// TwinCAT 3 PLC project task1
// ProgramVersion: 3.1.4022.4
// libraries:
//   Tc2_Standard, * (Beckhoff Automation GmbH)
//   Tc2_System, * (Beckhoff Automation GmbH)
//   Tc3_Module, * (Beckhoff Automation GmbH)
// project tree:
//   / PlcTask.TcTTO
//   POUs/ FB1.TcPOU, FB2.TcPOU, FB3.TcPOU, FB4.TcPOU, iFb.TcIO, MAIN.TcPOU
// real-time tasks:
//   TASK PlcTask: cycle T#10ms, priority 20, ADS port 350

CONFIGURATION task1
    RESOURCE PLC ON TwinCAT3
        TASK PlcTask(INTERVAL := T#10ms, PRIORITY := 20);
    END_RESOURCE
END_CONFIGURATION

// ---- POUs/iFb.TcIO
//Contiene due proprietà che sono i valori di input
//ed un metodo generico che calcola il valore
INTERFACE iFb

PROPERTY PUBLIC fInput1 : REAL
GET
END_GET
SET
END_SET
END_PROPERTY

PROPERTY PUBLIC fInput2 : REAL
GET
END_GET
SET
END_SET
END_PROPERTY

METHOD returnValue : REAL
VAR_INPUT
END_VAR
END_METHOD

END_INTERFACE

// ---- POUs/FB1.TcPOU
//La FB1 Implementa l'interfaccia iFB

FUNCTION_BLOCK PUBLIC FB1 IMPLEMENTS iFb
VAR_INPUT
END_VAR
VAR_OUTPUT
END_VAR
VAR
	fInternalInput1 : REAL;
	fInternalInput2 : REAL;
END_VAR

;

{warning 'add property implementation'}
PROPERTY fInput1 : REAL
GET
fInput1 := this^.fInternalInput1;
END_GET
SET
this^.fInternalInput1 := fInput1;
END_SET
END_PROPERTY

{warning 'add property implementation'}
PROPERTY fInput2 : REAL
GET
fInput2 := this^.fInternalInput2;
END_GET
SET
this^.fInternalInput2 := fInput2;
END_SET
END_PROPERTY

{warning 'add method implementation'}
METHOD returnValue : REAL
//Implementazione Interfaccia con somma
returnValue := this^.fInput1 + this^.fInput2;
END_METHOD

END_FUNCTION_BLOCK

// ---- POUs/FB2.TcPOU
//Anche FB2 Implementa l'interfaccia iFB
//Posso considerarla come un'altra implementazione della stessa

FUNCTION_BLOCK PUBLIC FB2 IMPLEMENTS iFb
VAR_INPUT
END_VAR
VAR_OUTPUT
END_VAR
VAR
	fInternalInput1 : REAL;
	fInternalInput2 : REAL;
END_VAR

{warning 'add property implementation'}
PROPERTY fInput1 : REAL
GET
fInput1 := this^.fInternalInput1;
END_GET
SET
this^.fInternalInput1 := fInput1;
END_SET
END_PROPERTY

{warning 'add property implementation'}
PROPERTY fInput2 : REAL
GET
fInput2 := this^.fInternalInput2;
END_GET
SET
this^.fInternalInput2 := fInput2;
END_SET
END_PROPERTY

{warning 'add method implementation'}
METHOD returnValue : REAL
//Implementazione Interfaccia con moltiplicazione
returnValue := this^.fInput1 * this^.fInput2;
END_METHOD

END_FUNCTION_BLOCK

// ---- POUs/FB3.TcPOU
//La FB3 estende la FB1 quindi anche lei implementa l'interfaccia  
//non devo però implementare i metodi get e set delle proprietà
FUNCTION_BLOCK FB3 EXTENDS FB1
VAR_INPUT
	bFlag : bool;
END_VAR
VAR_OUTPUT
END_VAR
VAR
END_VAR

{warning 'add method implementation'}
METHOD returnValue : REAL
//Estensione della funzione base
IF bFlag THEN
	returnValue := SUPER^.returnValue(); //Uso il metodo "padre"
ELSE
	returnValue := 0;		
END_IF
END_METHOD

END_FUNCTION_BLOCK

// ---- POUs/FB4.TcPOU
FUNCTION_BLOCK FB4
VAR_INPUT
	fbGenericFB : iFb;
	fInput1: REAL;
	fInput2: REAL; 
END_VAR
VAR_OUTPUT
	bIsEven : BOOL;
END_VAR
VAR
	iResult : INT;
END_VAR


//Inizializzo e uso la FB Generica grazie all'interfaccia
fbGenericFB.fInput1 := fInput1;
fbGenericFB.fInput2 := fInput2;

iResult := REAL_TO_INT(fbGenericFB.returnValue());

//Calcolo l'output
bIsEven := (iResult MOD 2) = 0;

END_FUNCTION_BLOCK

// ---- POUs/MAIN.TcPOU
PROGRAM MAIN
VAR
	//Input uguali per tutti
	fI1 : REAL := 5; 	
	fI2 : REAL := 2;
	
	//Le funzioni generiche FB4 che hanno in input una iFB
	fb4_1 : FB4;
	fb4_2 : FB4;
	fb4_3 : FB4;

	//Implementazioni di IFB
	fb1: FB1;		
	fb2: FB2;		
	fb3: FB3;
	bFlagFb3 :  BOOL;	
	
	//Risultati
	bResFB4_1 : BOOL;
	bResFB4_2 : BOOL;
	bResFB4_3 : BOOL;
END_VAR

//Passo il parametro in input a FB3 (non previsto dall'interfaccia)
fb3.bFlag := bFlagFb3;

//Uso la FB4 tre volte e richiamo 3 FB diverse che implementano la stessa interfaccia
fb4_1(fbGenericFB := fb1, fInput1 := fI1, fInput2 := fI2);
fb4_2(fbGenericFB := fb2, fInput1 := fI1, fInput2 := fI2);
fb4_3(fbGenericFB := fb3, fInput1 := fI1, fInput2 := fI2);

//Risultati
bResFB4_1 := fb4_1.bIsEven;  // Somma quindi 5 + 2 = 7 => False
bResFB4_2 := fb4_2.bIsEven;  // Moltiplicazione quindi 5 * 2 = 10 => True
bResFB4_3 := fb4_3.bIsEven;  // Se il flag è FALSE, => True, Se il flag è TRUE allora esgue la somma quindi 5 * 2 = 10 => True

END_PROGRAM
